// TIA Portal V20 export
ORGANIZATION_BLOCK "DiagnosticErrorInterrupt"   // OB82, SCL, DiagnosticErrorInterrupt
{ S7_Optimized_Access := 'TRUE' }
// stored: SetENOAutomatically false
   VAR_INPUT
      IO_State : Word;   // IO state of the HW object
      LADDR : HW_ANY;   // Hardware identifier
      Channel : UInt;   // Channel number
      MultiError : Bool;   // =true if more than one error is present
   END_VAR
BEGIN
   REGION Description head
       //==================================================================================
       // POSALUX Swiss SA / (C) Copyright 2025
       //----------------------------------------------------------------------------------
       // Title: DiagnosticErrorInterrupt
       // Comment/Function: Executes when the CPU detects a diagnostic error,
       //                   or if a diagnostics-capable module recognizes an error
       // Author: Fabien WALDT
       // Engineering: TIA Portal v19
       //----------------------------------------------------------------------------------
       // Change log table:
       // Version  | Date     | Expert in charge | Changes applied
       //----------------------------------------------------------------------------------
       // 00.00.01 | 20250423 | WFA              | First released version
       //==================================================================================
   END_REGION
END_ORGANIZATION_BLOCK
